Universal Robots PolyScope program: Demoprogramm.urp

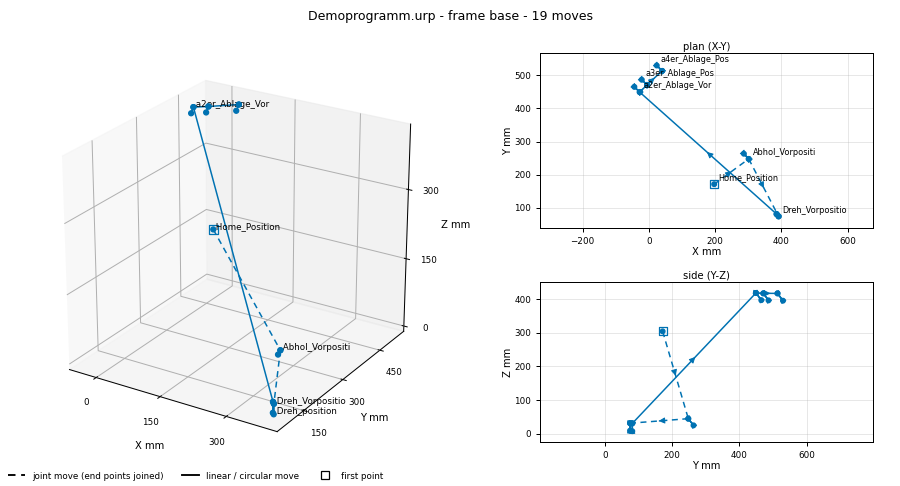
[picture p0: tool path of Demoprogramm.urp in frame base, 19 of 19 moves have a stored position in this frame; points joined in program order, loops and branches not executed]
ProgramRoot setBeforeStartSequence=true; directory=/programs/BoGieBae; kinematics=(a=[0, -0.425, -0.39225, 0, 0, 0], d=[0.08916, 0, 0, 0.10915, 0.09465, 0.0823], alpha=[1.5708, 0, 0, 1.5708, -1.5708, 0], deltaTheta=[0, 0, 0, 0, 0, 0], status=notInitialized); name=Demoprogramm; programVersion=(project__name=PolyScope, major__version=1, minor__version=8, svn__revision=25319, build__date=Oct 19 2016, 16:34:22); robotEnvironmentFileName=Modbus_Einstellungen; serialNumberRobot=2013215024
  BeforeStart description=COMMAND_SEQUENCE_BEFORE_PROGRAM_START; name=BeforeStart
    Script type=1; cachedFileContents=def gripper_init():
      |   i = 0
      |   iStep = 10
      |   while (iStep < 100) and (i < 20):
      |     if iStep == 10:
      |       if bit_of_word(modbus_get_signal_status("StatusWord", False), 6):
      |         modbus_set_output_register("ControlWord", 1, False)
      |         iStep = 20
      |       end
      |     end
      | 
      |     if iStep == 20:
      |       if bit_of_word(modbus_get_signal_status("StatusWord", False), 12):
      |         modbus_set_output_register("ControlWord", 0, False)
      |         iStep = 30
      |       end
      |     end
      | 
      |     if iStep == 30:
      |       if not bit_of_word(modbus_get_signal_status("StatusWord", False), 12):
      |         modbus_set_output_register("DeviceMode_Work", 25600, False)
      |         modbus_set_output_register("GripForce_Posit", 276, False)
      |         modbus_set_output_register("ControlWord", 1, False)
      |         iStep = 40
      |       end
      |     end
      | 
      | 
      |     if iStep == 40:
      |       if bit_of_word(modbus_get_signal_status("StatusWord", False), 12):
      |         modbus_set_output_register("ControlWord", 0, False)
      |         iStep = 100
      |       end
      |     end
      | 
      |     i = i + 1
      |     sleep(0.1)
      |   end
      |   if i >= 20:
      |     popup("Could not initialize gripper. Check the electrical connection and diagnosis word for more information.", title = "Error from Gripper", error = True, blocking = True)
      |   end
      | end
      | 
      | def bit_of_word(word, bit_number):
      |   return floor(word / pow(2, bit_number)) % 2 != 0
      | end
      | 
      | def gripper_open():
      |   modbus_set_output_register("ControlWord", 256, False)
      | end
      | 
      | def gripper_close():
      |   modbus_set_output_register("ControlWord", 512, False)
      | end
      | 
      | def gripper_reset_direction_flag():
      |   modbus_set_output_register("ControlWord", 4, False)
      |   i = 0
      |   while (not bit_of_word(modbus_get_signal_status("StatusWord", False), 13)) and (not bit_of_word(modbus_get_signal_status("StatusWord", False), 14)) and (i < 100):
      |     sleep(0.01)
      |     i = i + 1
      |   end
      |   if i >= 100:
      |     varmsg("Gripper Message", "Could not reset the direction flag.")
      |   end
      | end
      | 
      | def gripper_is_base_position():
      |   return bit_of_word(modbus_get_signal_status("StatusWord", False), 8)
      | end
      | 
      | def gripper_is_teach_position():
      |   return bit_of_word(modbus_get_signal_status("StatusWord", False), 9)
      | end
      | 
      | def gripper_is_work_position():
      |   return bit_of_word(modbus_get_signal_status("StatusWord", False), 10)
      | end
      | 
      | def gripper_get_actual_position():
      |   positionWord = modbus_get_signal_status("ActualPosition", False)
      |   return positionWord
      | end
      | 
      | def gripper_write_recipe(device_mode, workpiece_number, position_tolerance, grip_force, teach_position):
      |   modbus_set_output_register("DeviceMode_Work", (device_mode * 256 + workpiece_number), False)
      |   modbus_set_output_register("GripForce_Posit", (grip_force * 256 + position_tolerance), False)
      |   modbus_set_output_register("TeachPosition", teach_position, False)
      |   i = 0
      |   iStep = 10
      |   while (iStep < 100) and (i < 20):
      |     if iStep == 10:
      |       modbus_set_output_register("ControlWord", 1, False)
      |       iStep = 20
      |     end
      | 
      |     if iStep == 20:
      |       if bit_of_word(modbus_get_signal_status("StatusWord", False), 12):
      |         modbus_set_output_register("ControlWord", 0, False)
      |         iStep = 30
      |       end
      |     end
      | 
      |     if iStep == 30:
      |       if not bit_of_word(modbus_get_signal_status("StatusWord", False), 12):
      |         modbus_set_output_register("ControlWord", 2, False)
      |         iStep = 40
      |       end
      |     end
      | 
      |     if iStep == 40:
      |       if bit_of_word(modbus_get_signal_status("StatusWord", False), 12):
      |         modbus_set_output_register("ControlWord", 0, False)
      |         iStep = 50
      |       end
      |     end
      | 
      |     if iStep == 50:
      |       sleep(1)
      |       if not bit_of_word(modbus_get_signal_status("StatusWord", False), 12):
      |         iStep = 100
      |       end
      |     end
      |     i = i + 1
      |     sleep(0.1)
      |   end
      |   if i >= 20:
      |     varmsg("Gripper Message", "Could not write recipe.")
      |   end
      | end
      | 
      | def gripper_load_recipe(device_mode, workpiece_number):
      |   i = 0
      |   iStep = 10
      |   while (iStep < 100) and (i < 20):
      |     if iStep == 10:
      |       modbus_set_output_register("DeviceMode_Work", (device_mode * 256 + workpiece_number), False)
      |       iStep = 20
      |     end
      | 
      |     if iStep == 20:
      |       modbus_set_output_register("ControlWord", 1, False)
      |       iStep = 30
      |     end
      | 
      |     if iStep == 30:
      |       if bit_of_word(modbus_get_signal_status("StatusWord", False), 12):
      |         modbus_set_output_register("ControlWord", 0, False)
      |         iStep = 40
      |       end
      |     end
      | 
      |     if iStep == 40:
      |       if not bit_of_word(modbus_get_signal_status("StatusWord", False), 12):
      |         iStep = 100
      |       end
      |     end
      |     i = i + 1
      |     sleep(0.1)
      |   end
      |   if i >= 20:
      |     varmsg("Gripper Message", "Could not load recipe.")
      |   end
      | end
      | 
      | gripper_init(); scriptFile=/programs/BoGieBae/scripts/GEP2000.script
    Script type=0; expressionBranchNode=gripper_write_recipe(100, 1, 30, 2, 1754)
    Script type=0; expressionBranchNode=gripper_open()
    Wait analogComparison=0; analogInputRange=0; analogValue=0.0; digitalValue=0; selectedAnalogSensor=-1; selectedDigitalSensor=-1; waitTime=0.01; expr=gripper_is_base_position(); type=EXPRESSION_WAIT
  MainProgram cartesianAcceleration=1.2; cartesianSpeed=0.25; jointAcceleration=1.3962634015954636; jointSpeed=1.0471975511965976; moveAsFastAsPossible=true; sharedProcessMoveBlendRadius=0.025; featureReference=(installationNameReference=Base); motionType=JOINT_SPACE
    Suppressed suppressedNode=(MotionDefiningNode=(default=(cartesianAcceleration=1.2, cartesianSpeed=0.25, jointAcceleration=1.3962634015954636, jointSpeed=1.0471975511965976, moveAsFastAsPossible=true, sharedProcessMoveBlendRadius=0.025, standStillAtEnd=false, standStillAtStart=false, featureReference=(installationNameReference=Base), motionType=JOINT_SPACE)))
    Move cartesianAcceleration=1.2; cartesianSpeed=0.25; jointAcceleration=1.3962634015954636; jointSpeed=1.0471975511965976; moveAsFastAsPossible=true; sharedProcessMoveBlendRadius=0.025; featureReference=(installationNameReference=Base); motionType=JOINT_SPACE
      Waypoint blendRadius=0.1; cartesianAcceleration=1.2; cartesianSpeed=0.25; jointAcceleration=1.3962634015954636; jointSpeed=1.0471975511965976; nextMotionTime=2.0; useSharedParameters=true; position=TCP in base x=196.97 y=171.19 z=304.612 mm, rx=-2.4108 ry=1.9655 rz=-0.0013 rad; joints [195.457, -126.237, 116.935, -82.178, -89.008, 3.851] deg; positionType=FIXED_POSITION; waypointPoseInFeatureCoordinates=(pos=(x=0.19696954825323834, y=0.17119000264303585, z=0.3046121201739648), rot=(x=-2.4107908427795235, y=1.9654759359310756, z=-0.0013190025724868354)); name=Home_Position
    Move cartesianAcceleration=1.2; cartesianSpeed=0.25; jointAcceleration=1.3962634015954636; jointSpeed=1.0471975511965976; moveAsFastAsPossible=true; sharedProcessMoveBlendRadius=0.025; featureReference=(installationNameReference=Base); motionType=JOINT_SPACE
      Waypoint blendRadius=0.05; cartesianAcceleration=1.2; cartesianSpeed=0.25; jointAcceleration=1.3962634015954636; jointSpeed=1.0471975511965976; nextMotionTime=2.0; stoppoint=true; useSharedBlendParameter=true; useSharedParameters=true; position=TCP in base x=301.215 y=247.584 z=44.601 mm, rx=-2.4181 ry=0.9921 rz=1.0293 rad; joints [185.039, -82.358, 128.233, -102.559, -54.947, -51.138] deg; positionType=FIXED_POSITION; waypointPoseInFeatureCoordinates=(pos=(x=0.3012150352774236, y=0.24758389480715326, z=0.044600574159711234), rot=(x=-2.418143017531585, y=0.992146924823805, z=1.029344777209957)); name=Abhol_Vorpositi
    Move cartesianAcceleration=1.2; cartesianSpeed=0.02; jointAcceleration=1.3962634015954636; jointSpeed=1.0471975511965976; moveAsFastAsPossible=true; sharedProcessMoveBlendRadius=0.025; featureReference=(installationNameReference=Base); motionType=CARTESIAN_SPACE
      Waypoint blendRadius=0.05; cartesianAcceleration=1.2; cartesianSpeed=0.25; jointAcceleration=1.3962634015954636; jointSpeed=1.0471975511965976; nextMotionTime=2.0; stoppoint=true; useSharedBlendParameter=true; useSharedParameters=true; position=TCP in base x=286.716 y=263.089 z=24.691 mm, rx=-2.4182 ry=0.9921 rz=1.0294 rad; joints [187.444, -80.609, 130.859, -108.391, -53.651, -48.643] deg; positionType=FIXED_POSITION; waypointPoseInFeatureCoordinates=(pos=(x=0.28671560446139455, y=0.2630893704567889, z=0.024690725314600932), rot=(x=-2.418170308743977, y=0.9921498187414893, z=1.0293774766226786)); name=Abhol_Position
    Script type=0; expressionBranchNode=gripper_close()
    Wait analogComparison=0; analogInputRange=0; analogValue=0.0; digitalValue=0; selectedAnalogSensor=-1; selectedDigitalSensor=-1; waitTime=0.01; expr=gripper_is_teach_position(); type=EXPRESSION_WAIT
    Move cartesianAcceleration=1.2; cartesianSpeed=0.25; jointAcceleration=1.3962634015954636; jointSpeed=1.0471975511965976; moveAsFastAsPossible=true; sharedProcessMoveBlendRadius=0.025; featureReference=(installationNameReference=Base); motionType=CARTESIAN_SPACE
      Waypoint blendRadius=0.05; cartesianAcceleration=1.2; cartesianSpeed=0.25; jointAcceleration=1.3962634015954636; jointSpeed=1.0471975511965976; nextMotionTime=2.0; stoppoint=true; useSharedBlendParameter=true; useSharedParameters=true; position=TCP in base x=301.215 y=247.584 z=44.601 mm, rx=-2.4181 ry=0.9921 rz=1.0293 rad; joints [185.039, -82.358, 128.233, -102.559, -54.947, -51.138] deg; positionType=FIXED_POSITION; waypointPoseInFeatureCoordinates=(pos=(x=0.3012150352774236, y=0.24758389480715326, z=0.044600574159711234), rot=(x=-2.418143017531585, y=0.992146924823805, z=1.029344777209957)); name=Abhol_Vorpositi
    Move cartesianAcceleration=1.2; cartesianSpeed=0.25; jointAcceleration=1.3962634015954636; jointSpeed=1.0471975511965976; moveAsFastAsPossible=true; sharedProcessMoveBlendRadius=0.025; featureReference=(installationNameReference=Base); motionType=JOINT_SPACE
      Waypoint blendRadius=0.05; cartesianAcceleration=1.2; cartesianSpeed=0.25; jointAcceleration=1.3962634015954636; jointSpeed=1.0471975511965976; nextMotionTime=2.0; stoppoint=true; useSharedBlendParameter=true; useSharedParameters=true; position=TCP in base x=391.483 y=74.181 z=31.012 mm, rx=2.8689 ry=-1.2649 rz=-0.0098 rad; joints [174.942, -86.703, 134.032, -136.875, -90.221, -47.471] deg; positionType=FIXED_POSITION; waypointPoseInFeatureCoordinates=(pos=(x=0.3914830404452107, y=0.07418053055159589, z=0.031011839900466822), rot=(x=2.8689044644645754, y=-1.2649320757780709, z=-0.009753894932898795)); name=Dreh_Vorpositio
    Move cartesianAcceleration=1.2; cartesianSpeed=0.02; jointAcceleration=1.3962634015954636; jointSpeed=1.0471975511965976; moveAsFastAsPossible=true; sharedProcessMoveBlendRadius=0.025; featureReference=(installationNameReference=Base); motionType=CARTESIAN_SPACE
      Waypoint blendRadius=0.05; cartesianAcceleration=1.2; cartesianSpeed=0.25; jointAcceleration=1.3962634015954636; jointSpeed=1.0471975511965976; nextMotionTime=2.0; stoppoint=true; useSharedBlendParameter=true; useSharedParameters=true; position=TCP in base x=391.304 y=74.113 z=8.769 mm, rx=2.8689 ry=-1.2649 rz=-0.0099 rad; joints [174.929, -83.514, 135.402, -141.434, -90.221, -47.484] deg; positionType=FIXED_POSITION; waypointPoseInFeatureCoordinates=(pos=(x=0.3913043388812179, y=0.07411291985812235, z=0.008768688616671554), rot=(x=2.8688905645238156, y=-1.2649085807522824, z=-0.009863450518463058)); name=Dreh_position
    Script type=0; expressionBranchNode=gripper_open()
    Wait analogComparison=0; analogInputRange=0; analogValue=0.0; digitalValue=0; selectedAnalogSensor=-1; selectedDigitalSensor=-1; waitTime=0.01; expr=gripper_is_base_position(); type=EXPRESSION_WAIT
    Move cartesianAcceleration=1.2; cartesianSpeed=0.25; jointAcceleration=1.3962634015954636; jointSpeed=1.0471975511965976; moveAsFastAsPossible=true; sharedProcessMoveBlendRadius=0.025; featureReference=(installationNameReference=Base); motionType=CARTESIAN_SPACE
      Waypoint blendRadius=0.05; cartesianAcceleration=1.2; cartesianSpeed=0.25; jointAcceleration=1.3962634015954636; jointSpeed=1.0471975511965976; nextMotionTime=2.0; stoppoint=true; useSharedBlendParameter=true; useSharedParameters=true; position=TCP in base x=391.483 y=74.181 z=31.012 mm, rx=2.8689 ry=-1.2649 rz=-0.0098 rad; joints [174.942, -86.703, 134.032, -136.875, -90.221, -47.471] deg; positionType=FIXED_POSITION; waypointPoseInFeatureCoordinates=(pos=(x=0.3914830404452107, y=0.07418053055159589, z=0.031011839900466822), rot=(x=2.8689044644645754, y=-1.2649320757780709, z=-0.009753894932898795)); name=Dreh_Vorpositio
    Move cartesianAcceleration=1.2; cartesianSpeed=0.25; jointAcceleration=1.7453292519943295; jointSpeed=1.7453292519943295; moveAsFastAsPossible=true; sharedProcessMoveBlendRadius=0.025; featureReference=(installationNameReference=Base); motionType=JOINT_SPACE
      Waypoint blendRadius=0.007; cartesianAcceleration=1.2; cartesianSpeed=0.25; jointAcceleration=1.3962634015954636; jointSpeed=1.0471975511965976; nextMotionTime=2.0; stoppoint=true; useSharedBlendParameter=true; useSharedParameters=true; position=TCP in base x=385.583 y=80.889 z=30.534 mm, rx=1.1021 ry=-2.9324 rz=0.0002 rad; joints [175.878, -87.228, 134.701, -137.009, -90.22, 44.686] deg; positionType=FIXED_POSITION; waypointPoseInFeatureCoordinates=(pos=(x=0.38558331431342774, y=0.08088903013181878, z=0.030533609186055678), rot=(x=1.1020897885095777, y=-2.932352044859857, z=1.8668805476092362E-4)); name=Mess_Vorpositio
    Move cartesianAcceleration=1.2; cartesianSpeed=0.02; jointAcceleration=1.3962634015954636; jointSpeed=1.0471975511965976; moveAsFastAsPossible=true; sharedProcessMoveBlendRadius=0.025; featureReference=(installationNameReference=Base); motionType=CARTESIAN_SPACE
      Waypoint blendRadius=0.05; cartesianAcceleration=1.2; cartesianSpeed=0.25; jointAcceleration=1.3962634015954636; jointSpeed=1.0471975511965976; nextMotionTime=2.0; stoppoint=true; useSharedBlendParameter=true; useSharedParameters=true; position=TCP in base x=385.391 y=80.821 z=7.277 mm, rx=1.102 ry=-2.9324 rz=0.0002 rad; joints [175.864, -83.839, 136.14, -141.837, -90.22, 44.672] deg; positionType=FIXED_POSITION; waypointPoseInFeatureCoordinates=(pos=(x=0.3853909032595994, y=0.08082059795173481, z=0.007276975427450283), rot=(x=1.1020133753556973, y=-2.9323928255531735, z=1.921888143607728E-4)); name=Mess_Position
    Script type=0; expressionBranchNode=gripper_close()
    Wait analogComparison=0; analogInputRange=0; analogValue=0.0; digitalValue=0; selectedAnalogSensor=-1; selectedDigitalSensor=-1; waitTime=1.0; type=TIMER_WAIT
    Assignment assignmentValueSource=0; expr=gripper_get_actual_position(); operatorValueType=INTEGER; valueSource=EXPRESSION; variable=(name=greif_position, prefersPersistentValue=false, requestANewUniqueName=false)
    Move cartesianAcceleration=1.2; cartesianSpeed=0.25; jointAcceleration=1.3962634015954636; jointSpeed=1.0471975511965976; moveAsFastAsPossible=true; sharedProcessMoveBlendRadius=0.025; featureReference=(installationNameReference=Base); motionType=CARTESIAN_SPACE
      Waypoint blendRadius=0.01; cartesianAcceleration=1.2; cartesianSpeed=0.25; jointAcceleration=1.3962634015954636; jointSpeed=1.0471975511965976; nextMotionTime=2.0; useSharedParameters=true; position=TCP in base x=385.583 y=80.889 z=30.534 mm, rx=1.1021 ry=-2.9324 rz=0.0002 rad; joints [175.878, -87.228, 134.701, -137.009, -90.22, 44.686] deg; positionType=FIXED_POSITION; waypointPoseInFeatureCoordinates=(pos=(x=0.38558331431342774, y=0.08088903013181878, z=0.030533609186055678), rot=(x=1.1020897885095777, y=-2.932352044859857, z=1.8668805476092362E-4)); name=Mess_Vorpositio
    If expr=(ExpressionVariableNode < 1784) and (ExpressionVariableNode > 1724); type=IF_NODE
      Move cartesianAcceleration=1.2; cartesianSpeed=0.25; jointAcceleration=1.3962634015954636; jointSpeed=1.0471975511965976; moveAsFastAsPossible=true; sharedProcessMoveBlendRadius=0.025; featureReference=(installationNameReference=Base); motionType=CARTESIAN_SPACE
        Waypoint blendRadius=0.05; cartesianAcceleration=1.2; cartesianSpeed=0.25; jointAcceleration=1.3962634015954636; jointSpeed=1.0471975511965976; nextMotionTime=2.0; stoppoint=true; useSharedBlendParameter=true; useSharedParameters=true; position=TCP in base x=-27.811 y=449.107 z=418.936 mm, rx=0.9731 ry=-2.4419 rz=-1.0328 rad; joints [240.671, -109.346, 103.976, -100.138, -45.67, 113.567] deg; positionType=FIXED_POSITION; waypointPoseInFeatureCoordinates=(pos=(x=-0.027811396833660174, y=0.4491070806637381, z=0.4189363462455312), rot=(x=0.9730971805514387, y=-2.4418625412619437, z=-1.0327672967853567)); name=a2er_Ablage_Vor
      Move cartesianAcceleration=1.2; cartesianSpeed=0.02; jointAcceleration=1.3962634015954636; jointSpeed=1.0471975511965976; moveAsFastAsPossible=true; sharedProcessMoveBlendRadius=0.025; featureReference=(installationNameReference=Base); motionType=CARTESIAN_SPACE
        Waypoint blendRadius=0.05; cartesianAcceleration=1.2; cartesianSpeed=0.25; jointAcceleration=1.3962634015954636; jointSpeed=1.0471975511965976; nextMotionTime=2.0; stoppoint=true; useSharedBlendParameter=true; useSharedParameters=true; position=TCP in base x=-43.847 y=464.918 z=397.5 mm, rx=0.9729 ry=-2.4419 rz=-1.0327 rad; joints [244.221, -107.458, 106.623, -107.93, -46.717, 118.269] deg; positionType=FIXED_POSITION; waypointPoseInFeatureCoordinates=(pos=(x=-0.04384653695087574, y=0.4649184309215718, z=0.39749956894322175), rot=(x=0.9729026178014861, y=-2.4419202262891253, z=-1.0326526348396754)); name=a2er_Ablage_Pos
      Script type=0; expressionBranchNode=gripper_open()
      Wait analogComparison=0; analogInputRange=0; analogValue=0.0; digitalValue=0; selectedAnalogSensor=-1; selectedDigitalSensor=-1; waitTime=0.01; expr=gripper_is_base_position(); type=EXPRESSION_WAIT
      Move cartesianAcceleration=1.2; cartesianSpeed=0.25; jointAcceleration=1.3962634015954636; jointSpeed=1.0471975511965976; moveAsFastAsPossible=true; sharedProcessMoveBlendRadius=0.025; featureReference=(installationNameReference=Base); motionType=CARTESIAN_SPACE
        Waypoint blendRadius=0.05; cartesianAcceleration=1.2; cartesianSpeed=0.25; jointAcceleration=1.3962634015954636; jointSpeed=1.0471975511965976; nextMotionTime=2.0; stoppoint=true; useSharedBlendParameter=true; useSharedParameters=true; position=TCP in base x=-27.811 y=449.107 z=418.936 mm, rx=0.9731 ry=-2.4419 rz=-1.0328 rad; joints [240.671, -109.346, 103.976, -100.138, -45.67, 113.567] deg; positionType=FIXED_POSITION; waypointPoseInFeatureCoordinates=(pos=(x=-0.027811396833660174, y=0.4491070806637381, z=0.4189363462455312), rot=(x=0.9730971805514387, y=-2.4418625412619437, z=-1.0327672967853567)); name=a2er_Ablage_Vor
    If expr=(ExpressionVariableNode < 994) and (ExpressionVariableNode > 934); type=ELSEIF_NODE
      Move cartesianAcceleration=1.2; cartesianSpeed=0.25; jointAcceleration=1.3962634015954636; jointSpeed=1.0471975511965976; moveAsFastAsPossible=true; sharedProcessMoveBlendRadius=0.025; featureReference=(installationNameReference=Base); motionType=CARTESIAN_SPACE
        Waypoint blendRadius=0.05; cartesianAcceleration=1.2; cartesianSpeed=0.25; jointAcceleration=1.3962634015954636; jointSpeed=1.0471975511965976; nextMotionTime=2.0; stoppoint=true; useSharedBlendParameter=true; useSharedParameters=true; position=TCP in base x=-5.862 y=471.012 z=417.713 mm, rx=0.973 ry=-2.4419 rz=-1.0328 rad; joints [239.37, -105.628, 101.362, -100.007, -45.335, 111.804] deg; positionType=FIXED_POSITION; waypointPoseInFeatureCoordinates=(pos=(x=-0.005862297981660286, y=0.47101151962530535, z=0.41771325663030995), rot=(x=0.9730461450336466, y=-2.441856659529699, z=-1.0327525073376624)); name=a3er_Ablage_Vor
      Move cartesianAcceleration=1.2; cartesianSpeed=0.02; jointAcceleration=1.3962634015954636; jointSpeed=1.0471975511965976; moveAsFastAsPossible=true; sharedProcessMoveBlendRadius=0.025; featureReference=(installationNameReference=Base); motionType=CARTESIAN_SPACE
        Waypoint blendRadius=0.05; cartesianAcceleration=1.2; cartesianSpeed=0.25; jointAcceleration=1.3962634015954636; jointSpeed=1.0471975511965976; nextMotionTime=2.0; stoppoint=true; useSharedBlendParameter=true; useSharedParameters=true; position=TCP in base x=-21.479 y=486.412 z=396.864 mm, rx=0.973 ry=-2.4418 rz=-1.0327 rad; joints [242.6, -103.908, 103.87, -107.261, -46.215, 116.142] deg; positionType=FIXED_POSITION; waypointPoseInFeatureCoordinates=(pos=(x=-0.021478674718793046, y=0.4864123744949015, z=0.3968636422591287), rot=(x=0.9730477232717049, y=-2.44182318950939, z=-1.0327496351967886)); name=a3er_Ablage_Pos
      Script type=0; expressionBranchNode=gripper_open()
      Wait analogComparison=0; analogInputRange=0; analogValue=0.0; digitalValue=0; selectedAnalogSensor=-1; selectedDigitalSensor=-1; waitTime=0.01; expr=gripper_is_base_position(); type=EXPRESSION_WAIT
      Move cartesianAcceleration=1.2; cartesianSpeed=0.25; jointAcceleration=1.3962634015954636; jointSpeed=1.0471975511965976; moveAsFastAsPossible=true; sharedProcessMoveBlendRadius=0.025; featureReference=(installationNameReference=Base); motionType=CARTESIAN_SPACE
        Waypoint blendRadius=0.05; cartesianAcceleration=1.2; cartesianSpeed=0.25; jointAcceleration=1.3962634015954636; jointSpeed=1.0471975511965976; nextMotionTime=2.0; stoppoint=true; useSharedBlendParameter=true; useSharedParameters=true; position=TCP in base x=-5.862 y=471.012 z=417.713 mm, rx=0.973 ry=-2.4419 rz=-1.0328 rad; joints [239.37, -105.628, 101.362, -100.007, -45.335, 111.804] deg; positionType=FIXED_POSITION; waypointPoseInFeatureCoordinates=(pos=(x=-0.005862297981660286, y=0.47101151962530535, z=0.41771325663030995), rot=(x=0.9730461450336466, y=-2.441856659529699, z=-1.0327525073376624)); name=a3er_Ablage_Vor
    If expr=(ExpressionVariableNode < 201) and (ExpressionVariableNode > 141); type=ELSEIF_NODE
      Move cartesianAcceleration=1.2; cartesianSpeed=0.25; jointAcceleration=1.3962634015954636; jointSpeed=1.0471975511965976; moveAsFastAsPossible=true; sharedProcessMoveBlendRadius=0.025; featureReference=(installationNameReference=Base); motionType=CARTESIAN_SPACE
        Waypoint blendRadius=0.05; cartesianAcceleration=1.2; cartesianSpeed=0.25; jointAcceleration=1.3962634015954636; jointSpeed=1.0471975511965976; nextMotionTime=2.0; stoppoint=true; useSharedBlendParameter=true; useSharedParameters=true; position=TCP in base x=40.047 y=513.255 z=417.653 mm, rx=0.9732 ry=-2.4419 rz=-1.0327 rad; joints [236.953, -98.163, 95.018, -98.779, -44.787, 108.479] deg; positionType=FIXED_POSITION; waypointPoseInFeatureCoordinates=(pos=(x=0.04004661610113262, y=0.5132549666749785, z=0.417653374881612), rot=(x=0.9731588992973493, y=-2.4418698570457757, z=-1.0326537157284101)); name=a4er_Ablage_Vor
      Move cartesianAcceleration=1.2; cartesianSpeed=0.02; jointAcceleration=1.3962634015954636; jointSpeed=1.0471975511965976; moveAsFastAsPossible=true; sharedProcessMoveBlendRadius=0.025; featureReference=(installationNameReference=Base); motionType=CARTESIAN_SPACE
        Waypoint blendRadius=0.05; cartesianAcceleration=1.2; cartesianSpeed=0.25; jointAcceleration=1.3962634015954636; jointSpeed=1.0471975511965976; nextMotionTime=2.0; stoppoint=true; useSharedBlendParameter=true; useSharedParameters=true; position=TCP in base x=23.662 y=529.423 z=395.855 mm, rx=0.9731 ry=-2.4417 rz=-1.033 rad; joints [239.94, -96.604, 97.552, -105.765, -45.479, 112.58] deg; positionType=FIXED_POSITION; waypointPoseInFeatureCoordinates=(pos=(x=0.023662388558847246, y=0.5294225888496282, z=0.39585495488520345), rot=(x=0.9731186617477213, y=-2.4417262393712873, z=-1.0329680793412046)); name=a4er_Ablage_Pos
      Script type=0; expressionBranchNode=gripper_open()
      Wait analogComparison=0; analogInputRange=0; analogValue=0.0; digitalValue=0; selectedAnalogSensor=-1; selectedDigitalSensor=-1; waitTime=0.01; expr=gripper_is_base_position(); type=EXPRESSION_WAIT
      Move cartesianAcceleration=1.2; cartesianSpeed=0.25; jointAcceleration=1.3962634015954636; jointSpeed=1.0471975511965976; moveAsFastAsPossible=true; sharedProcessMoveBlendRadius=0.025; featureReference=(installationNameReference=Base); motionType=CARTESIAN_SPACE
        Waypoint blendRadius=0.05; cartesianAcceleration=1.2; cartesianSpeed=0.25; jointAcceleration=1.3962634015954636; jointSpeed=1.0471975511965976; nextMotionTime=2.0; stoppoint=true; useSharedBlendParameter=true; useSharedParameters=true; position=TCP in base x=40.047 y=513.255 z=417.653 mm, rx=0.9732 ry=-2.4419 rz=-1.0327 rad; joints [236.953, -98.163, 95.018, -98.779, -44.787, 108.479] deg; positionType=FIXED_POSITION; waypointPoseInFeatureCoordinates=(pos=(x=0.04004661610113262, y=0.5132549666749785, z=0.417653374881612), rot=(x=0.9731588992973493, y=-2.4418698570457757, z=-1.0326537157284101)); name=a4er_Ablage_Vor
    If type=ELSE_NODE
      Popup haltProgram=true; message=Legogroesse konnte nicht zugeordnet werden.; type=WARNING
